// TIA Portal V17 export
// export: Created 2024-09-18T06:05:35.2359796Z, ExportSetting WithDefaults, DisplayName Totally Integrated Automation Portal, DisplayVersion V17, DisplayName TIA Portal Openness, DisplayVersion V17, DisplayName TIA Portal Version Control Interface, DisplayVersion V17, DisplayName STEP 7 Professional, DisplayVersion V17, DisplayName STEP 7 Safety, DisplayVersion V17, DisplayName WinCC Advanced / Unified PC, DisplayVersion V17
FUNCTION "Analog Input Scaling" : Void   // FC2, LAD
{ S7_Optimized_Access := 'TRUE' }
VERSION : 0.1
// stored: AutoNumber true, IsIECCheckEnabled false, SetENOAutomatically false, UDAEnableTagReadback false
   VAR_INPUT
      iNormMin : Int;
      iNormMax : Int;
      iValueInput : Int;
      "rScale Min" : Real;
      rScaleMax : Real;
   END_VAR
   VAR_OUTPUT
      rScaleOut : Real;
   END_VAR
   VAR_TEMP
      rNormTemp : Real;
   END_VAR
BEGIN

REGION Network 1
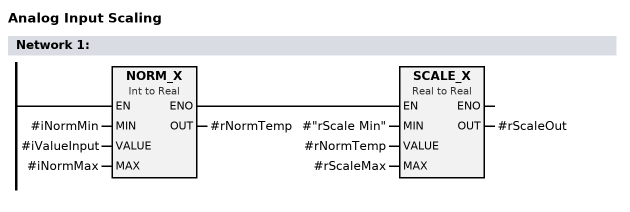
   RUNG wire#powerrail
      { S7_Templates := "[SrcType := Int, DestType := Real]" } Normalize(min := #iNormMin, value := #iValueInput, max := #iNormMax, out => #rNormTemp)
      { S7_Templates := "[SrcType := Real, DestType := Real]" } Scale(min := #"rScale Min", value := #rNormTemp, max := #rScaleMax, out => #rScaleOut)
   END_RUNG
   // the same network as SCL:
   #rNormTemp := NORM_X(MIN := #iNormMin, VALUE := #iValueInput, MAX := #iNormMax);
   #rScaleOut := SCALE_X(MIN := #"rScale Min", VALUE := #rNormTemp, MAX := #rScaleMax);
END_REGION
END_FUNCTION
